FUNCTION PackByte : INT
VAR_INPUT
	B0				: BOOL ;
	B1				: BOOL ;
	B2				: BOOL ;
	B3				: BOOL ;
	B4				: BOOL ;
	B5				: BOOL ;
	B6				: BOOL ;
	B7				: BOOL ;	
END_VAR
VAR
END_VAR

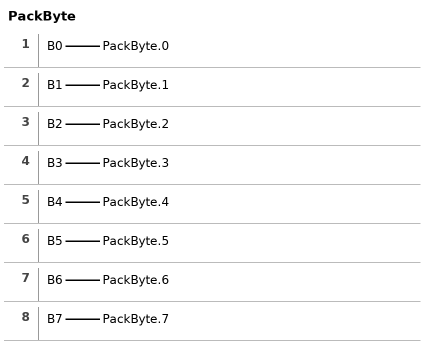
// NETWORK 1
PackByte.0 := B0;

// NETWORK 2
PackByte.1 := B1;

// NETWORK 3
PackByte.2 := B2;

// NETWORK 4
PackByte.3 := B3;

// NETWORK 5
PackByte.4 := B4;

// NETWORK 6
PackByte.5 := B5;

// NETWORK 7
PackByte.6 := B6;

// NETWORK 8
PackByte.7 := B7;

END_FUNCTION

(* stored: Version 1.1.0.1, ProductVersion 3.1.4026.18
   POU PackByte: Id {35d136b4-fb69-493c-96da-7f7401b2b3a2}, SpecialFunc None *)
